// TIA Portal V15.1 export
// export: Created 2024-05-17T05:38:43.7837693Z, ExportSetting WithDefaults, DisplayName Totally Integrated Automation Portal, DisplayVersion V15.1 Update 5, DisplayName TIA Portal Openness, DisplayVersion V15.1 Update 5, DisplayName SINAMICS Startdrive Advanced, DisplayVersion V15.1, DisplayName G130, G150, S120, S150, SINAMICS MV, S210, DisplayVersion V15.1, DisplayName G110M, G120, G120C, G120D, G120P, DisplayVersion V15.1, DisplayName STEP 7 Professional, DisplayVersion V15.1 Update 5, DisplayName STEP 7 Safety, DisplayVersion V15.1, DisplayName WinCC Professional, DisplayVersion V15.1 Update 5, DisplayName SIMATIC Visualization Architect, DisplayVersion V15.1
FUNCTION "LGBCalcOvertimeMoviPro" : Void   // FC6628, SCL
{ S7_Optimized_Access := 'TRUE' }
VERSION : 0.1
// stored: AutoNumber false, IsIECCheckEnabled false, SetENOAutomatically False, UDAEnableTagReadback false
   VAR_INPUT
      I_Speed : Real;   // Speed value in mm/s / High speed value 0-100%
      I_Diff_Pos : Real;   // Difference Positions Stop / Position Stop 1
      C_ProcAlm : Real;   // Procent for Alarm time
      C_Acceleration : Real;   // Acceleration in mm/s²
   END_VAR
   VAR_OUTPUT
      O_RunTimeMax : DInt;   // Overtime in millisec
   END_VAR
   VAR_TEMP
      Diff_Pos : Real;   // Difference Positions Stop / Position Stop 1
      Ramp : Real;   // Ramp in sec
      DistRamp : Real;   // Distance Ramp in mm
      DistSpeed : Real;   // Distance High speed in mm
      TimeSpeed : Real;   // Time High speed in sec
      RunTimeMax : Real;   // Overtime in sec
   END_VAR
BEGIN
   // LOGIC
   IF (#I_Speed <> 0.0) AND (#I_Diff_Pos <> 0.0) AND (#C_Acceleration <> 0.0) THEN
       // Ramp
       #Ramp := (#I_Speed / #C_Acceleration);

       // x = x0 + v0t + 1/2 * a * t² [mm]
       #DistRamp := 0 + 0 + (0.5 * #C_Acceleration * #Ramp * #Ramp);
   ELSE
       #Ramp := 0.0;
       #DistRamp := 0.0;
   END_IF;

   IF (#I_Diff_Pos >= 0.0) THEN
       #Diff_Pos := #I_Diff_Pos;
   ELSE
       #Diff_Pos:= (#I_Diff_Pos * -1.0);
   END_IF;

   #DistSpeed := #Diff_Pos - #DistRamp - #DistRamp;
   #TimeSpeed := (#DistSpeed /#I_Speed);

   IF (#Diff_Pos <> 0.0) THEN
       #RunTimeMax := #Ramp + #TimeSpeed + #Ramp;
       #RunTimeMax := (#RunTimeMax * (#C_ProcAlm / 100.0)) + #RunTimeMax;
   ELSE
       #RunTimeMax := 0.0;
   END_IF;

   // OUTPUT
   #O_RunTimeMax := REAL_TO_DINT(#RunTimeMax * 1000.0);
END_FUNCTION
